// TIA Portal V20 export
DATA_BLOCK "HmiInterface"   // DB92
// stored: Access Published, MemoryReserve 100, Namespace Unit1.Em9
   VAR
      em : "LAF_typeEmInterface";
      vision : "LER_typeSequenceInterface";
      GRnR_vision { S7_SetPoint := 'True'} : "LER_typeSequenceInterface";
      cmVisionJRDetect : "LBC_typeDigitalSignalInterface";
      cmVisionStageLiftUpDown : "LBC_typeTwoWayActuatorInterface";
      cmVisionLightUpDown : "LBC_typeTwoWayActuatorInterface";
      cmVisionControl : "LER_typeVisionInterface";
      cmVisionConvertData : "LER_typeVisionResultData";
   END_VAR
   VAR RETAIN
      cmVisionHistory : "LER_typeVisionHistory";
      "cmVisionHistory_r&r" : "LER_typeVisionHistory";
   END_VAR
   VAR
      VisionNgAlarmCount { S7_SetPoint := 'True'} : "LER_typeAlarmCounterInterface";
      gaugeRnR : "Unit1.Em9.typeGaugeRnRHmiInterface";
      intCondition : "Unit1.Em9.typeIntConditionHmiInterface";
      VisionRetryCount : "Unit1.Em9.typeVisionRetryHmiInterface";
      VisionResultNG : Bool;
      VisionResultOK : Bool;
      VisionRetryReset : Bool;
   END_VAR
BEGIN
   VisionNgAlarmCount.referenceDesignator := WSTRING#'Em9 Vision Ng Alarm Count';
END_DATA_BLOCK
